// TIA Portal V20 export
DATA_BLOCK "ConveyorMotor1"   // DB4
// stored: InstanceOfName MotorDOL, InstanceOfType FB
"MotorDOL"
   // VAR RETAIN
   //    IO { S7_SetPoint := 'True'} : "TypeDOL";
   // END_VAR
   // VAR
   //    FaultTripTimer2 { S7_SetPoint := 'True'} : TON_TIME;
   // END_VAR
BEGIN
   IO.InHand := FALSE;
END_DATA_BLOCK
